Fanuc KAREL source: kt00133.KL

-- PROVISIONAL review KL for V1013-1; original PC SHA256 542356148e7a6f4b66dd595f3b758ce19be1c8b7b6ad503ca2002a3279ffab6f
-- Incomplete behavior may be omitted. Consult companion uncertainty JSON. Do not deploy.
PROGRAM KT00133
%NOLOCKGROUP
VAR
  I1 : INTEGER
  OUT : INTEGER
-- UNRESOLVED_DECL Y2 type=002018
BEGIN
  -- UNRESOLVED_PC offsets 5-16; opcodes 2E,23
  -- UNRESOLVED_PC offsets 21-35; opcodes 2E,22,9D,33,B2
  -- UNRESOLVED_PC offsets 40-62; opcodes 21,22,9D,33,B1,55,23
  -- UNRESOLVED_PC offsets 67-71; opcodes 7F
END KT00133
